Staubli VAL3: JTrajPtFullBody.pjx

--- JTrajPtFullBody.pjx ---
Parameters version=s7.3 stackSize=5000 millimeterUnit=true
Program file=start.pgx
Program file=stop.pgx
Data file=JTrajPtFullBody.dtx

--- JTrajPtFullBody.dtx ---
public num accelerations[10]
public num positions[10]
public num robotId
public num sequence
public num time
public num validFields
public num velocities[10]

--- start.pgx ---
program start()
begin
end
